SUBAPPLICATION logiBUS_AI_IDA_OPC (* logiBUS_AI_IDA (Analog-Eingang) auf VT-Zahlenfeld (Rohwert+Prozent, geteilte CNumberVariable) + Bargraph + OPC-UA (Rohwert DWORD + Prozent REAL, generisch, ein Kanal) *)
  (* Standard: 61499-2; Description: Copyright (c) 2026 Meisterschulen am Ostbahnhof This program and the accompanying materials are made available under the terms of the Eclipse Public License 2.0 which is available at https://www.eclipse.org/legal/epl-2.0/ SPDX-License-Identifier: EPL-2.0 *)
  (* Version 1.0, 2026-08-30, Franz Höpfinger, Meisterschulen am Ostbahnhof, initial API and implementation and/or initial documentation *)
  PACKAGE MyLib::sys;
  IMPORT isobus::UT::Q::const::IDs::ID_NULL;
  IMPORT logiBUS::io::AI::logiBUS_AI;
  IMPORT logiBUS::io::AI::logiBUS_AI_S;
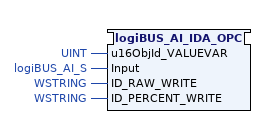
  VAR_INPUT
    u16ObjId_VALUEVAR : UINT := ID_NULL; (* Object ID CNumberVariable (Rohwert 0-4095, gemeinsam gebunden an Rohwert-Zahlenfeld, Prozent-Zahlenfeld und Bargraph - Prozent/Bargraph nutzen ihre eigene VT-Scale auf denselben Rohwert) *)
    Input : logiBUS::io::AI::logiBUS_AI_S := logiBUS_AI::Invalid; (* Identify the Input AnalogInput_I1..I8 *)
    ID_RAW_WRITE : WSTRING; (* Rohwert-Ruckmelde-Adresse (DWORD 0-4095, ACTION=PUBLISH) *)
    ID_PERCENT_WRITE : WSTRING; (* Prozent-Ruckmelde-Adresse (REAL 0.0-100.0, ACTION=PUBLISH, linear ohne physikalische Kalibrierung) *)
  END_VAR
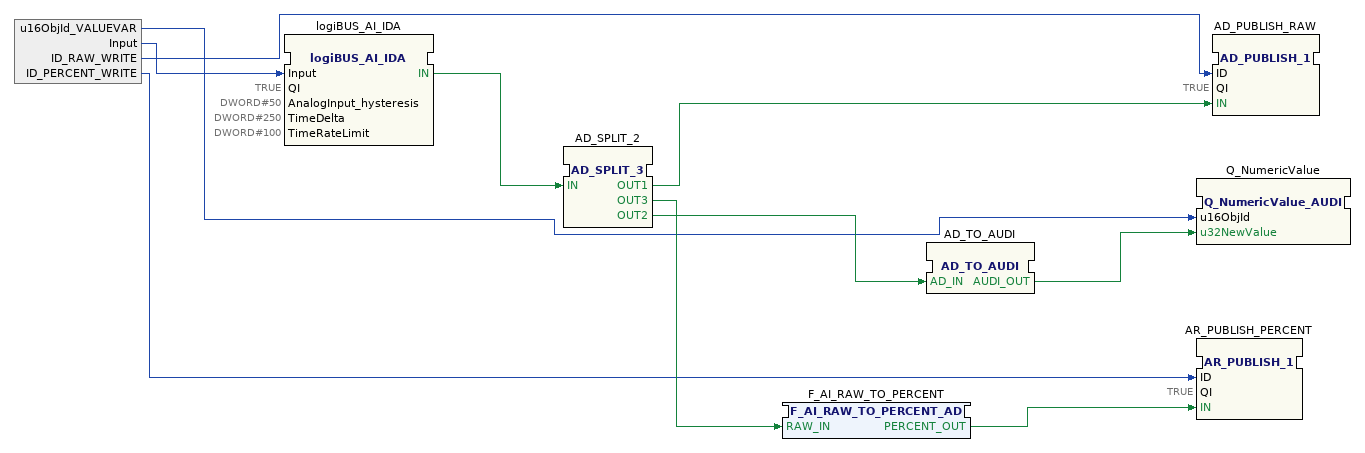
  FBS
    logiBUS_AI_IDA : logiBUS::io::AI::logiBUS_AI_IDA(QI := TRUE, AnalogInput_hysteresis := DWORD#50, TimeDelta := DWORD#250, TimeRateLimit := DWORD#100);
    AD_SPLIT_2 : adapter::events::unidirectional::AD_SPLIT_3;
    AD_PUBLISH_RAW : adapter::net::AD_PUBLISH_1(QI := TRUE);
    Q_NumericValue : isobus::UT::Q::Q_NumericValue_AUDI;
    AR_PUBLISH_PERCENT : adapter::net::AR_PUBLISH_1(QI := TRUE);
    AD_TO_AUDI : adapter::conversion::unidirectional::AD_TO_AUDI;
  END_FBS
  SUBAPPS
    F_AI_RAW_TO_PERCENT : MyLib::sys::F_AI_RAW_TO_PERCENT_AD;
  END_SUBAPPS
  DATA_CONNECTIONS
    Input TO logiBUS_AI_IDA.Input;
    u16ObjId_VALUEVAR TO Q_NumericValue.u16ObjId;
    ID_RAW_WRITE TO AD_PUBLISH_RAW.ID;
    ID_PERCENT_WRITE TO AR_PUBLISH_PERCENT.ID;
  END_CONNECTIONS
  ADAPTER_CONNECTIONS
    logiBUS_AI_IDA.IN TO AD_SPLIT_2.IN;
    AD_SPLIT_2.OUT1 TO AD_PUBLISH_RAW.IN;
    AD_SPLIT_2.OUT3 TO F_AI_RAW_TO_PERCENT.RAW_IN;
    F_AI_RAW_TO_PERCENT.PERCENT_OUT TO AR_PUBLISH_PERCENT.IN;
    AD_TO_AUDI.AUDI_OUT TO Q_NumericValue.u32NewValue;
    AD_SPLIT_2.OUT2 TO AD_TO_AUDI.AD_IN;
  END_CONNECTIONS
END_SUBAPPLICATION
